// An enum that can be used to represent getters and setters.
{attribute 'qualified_only'}
{attribute 'to_string'}
TYPE E_Accessor :
(
	_ := 0, // Unknown/Invalid
	Get,
	Set
)BYTE;
END_TYPE

(* stored: Version 1.1.0.1
   EnumerationTextList E_Accessor: Id {c59c5995-9ee9-07ff-0331-8bb2064d0e78} *)
